# B&R Automation Studio project CNC_Machine_5_18
Automation Studio 4.12.2.93; technology packages: mapp 5.18.0, mappMotion 5.18.1, mappView 5.18.1

## Configuration Config1

CPU X20CP1586, AutomationRuntime C4.73, Build 4.1.2, Vc V4.72.0

### Task classes (Cpu.sw)
```
Cyclic#1:
  Program <- Program.prg
DataObjects: McAcpSys
NcDataObjects: CncProg <- CNCProg.CncProg.dob, McDriveLog
Binaries: McAcpDrv, udbdef, McAcpSim, mvLoader, arflatprv, TCData, OpcUaSrv, McMechSys, FWRules, arcoal, arsvcreg, iomap, asfw, Config_3, Config_4, Role, ashwac, Hierarchy, sysconf, Config_2, arconfig, Config_1, ashwd, Config, User
Libraries: McBase, MpCnc, MpBase, McAxGroup, McPathGen, McAxis, McProgInt, McAcpAx, MpCodeBox, standard, FileIO, AsArLog, AsArProf, AsMem, DataObj, sys_lib, astime, runtime, MpFile, MpServer, MpDatabase, AsHttp, asieccon, asbrstr, asio, asepl, asusb, aruser, arssl, powerlnk, MpData, brsystem, MpAlarmX
```

### Hardware
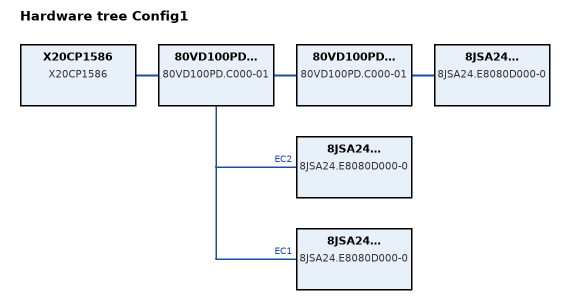
```
80VD100PD.C000-01 : 80VD100PD.C000-01 v2.5.0.0  [PLK1 -> X20CP1586.IF3 [Cable Type=PowerlinkCable, Length=10, Version=1.0.0.3]; PLK2 -> 80VD100PD.C000-01a.PLK2 [Cable Type=PowerlinkCable, Length=10, Version=1.0.0.3]; EC1 -> 8JSA24.E8080D000-0a.EC; EC2 -> 8JSA24.E8080D000-0.EC; MT2 -> 8JSA24.E8080D000-0.MT]
  DriveConfiguration/Module:
    McAcoposTypeID = AcoposMicroDConfig
    ActivateACOPOSSimulationOnPLC = 0
  DriveConfiguration/Channel[1]/RealAxis:
    AxisReference = gAxisQX
    MechanicalElementsIsInvisible = 0
  DriveConfiguration/Channel[1]/RealAxis/MechanicalElements/Gearbox:
    InputIsReadOnly = 0
    Input = 1
    OutputIsReadOnly = 0
    Output = 1
  DriveConfiguration/Channel[1]/RealAxis/MechanicalElements/RotaryToLinearTransformation:
    ReferenceDistanceIsReadOnly = 0
    ReferenceDistance = 1
  DriveConfiguration/Channel[1]/RealAxis/Controller:
    ModeIsReadOnly = 0
    Mode = PositionController
  DriveConfiguration/Channel[1]/RealAxis/Controller/Mode/Position:
    ProportionalGain = 50.0
    IntegrationTime = 0.0
    PredictionTime = 0.0004
    TotalDelayTime = 0.0004
  DriveConfiguration/Channel[1]/RealAxis/Controller/Mode/Speed:
    ProportionalGainIsReadOnly = 0
    ProportionalGain = 2.0
    IntegrationTimeIsReadOnly = 0
    IntegrationTime = 0.0
    FilterTimeIsReadOnly = 0
    FilterTime = 0.0
  DriveConfiguration/Channel[1]/RealAxis/Controller/Mode/LoopFilters:
    LoopFilterXIsReadOnly = 0
    LoopFilter1 = NotUsed
    LoopFilter2 = NotUsed
    LoopFilter3 = NotUsed
  DriveConfiguration/Channel[1]/RealAxis/Homing:
    ModeIsReadOnly = 0
    Mode = Direct
  DriveConfiguration/Channel[1]/RealAxis/Homing/Mode:
    Position = 0.0
    ReferencePulse = NotUsed
  DriveConfiguration/Channel[1]/RealAxis/Homing:
    RestorePositionVariable = 
  DriveConfiguration/Channel[1]/RealAxis/StopReaction:
    QuickstopIsReadOnly = 0
    Quickstop = DecelerationLimit
    DriveErrorIsReadOnly = 0
    DriveError = DecelerationLimit
  DriveConfiguration/Channel[1]/RealAxis/MovementErrorLimits:
    PositionError = 1.0
    VelocityErrorMonitoring = Automatic1
  DriveConfiguration/Channel[1]/RealAxis:
    JerkFilterIsReadOnly = 0
    JerkFilter = NotUsed
  DriveConfiguration/Channel[1]/RealAxis/DigitalInputs/HomingSwitch:
    SourceIsReadOnly = 0
    Source = NotUsed
    Level = High
  DriveConfiguration/Channel[1]/RealAxis/DigitalInputs/PositiveLimitSwitch:
    SourceIsReadOnly = 0
    Source = NotUsed
    Level = High
  DriveConfiguration/Channel[1]/RealAxis/DigitalInputs/NegativeLimitSwitch:
    SourceIsReadOnly = 0
    Source = NotUsed
    Level = High
  DriveConfiguration/Channel[1]/RealAxis/DigitalInputs/Trigger1:
    Source = X2Trigger1
    Level = High
  DriveConfiguration/Channel[1]/RealAxis/DigitalInputs/Trigger2:
    Source = X2Trigger2
    Level = High
  DriveConfiguration/Channel[1]/RealAxis/DigitalInputs/Quickstop:
    Input = Trigger2
  DriveConfiguration/Channel[1]/RealAxis/Simulation:
    SimulationModeOnPLC = SetValueGeneration
    SimulationModeOnACOPOS = NotUsed
  DriveConfiguration/Channel[2]/RealAxis:
    AxisReference = gAxisQY
    MechanicalElementsIsInvisible = 0
  DriveConfiguration/Channel[2]/RealAxis/MechanicalElements/Gearbox:
    InputIsReadOnly = 0
    Input = 1
    OutputIsReadOnly = 0
    Output = 1
  DriveConfiguration/Channel[2]/RealAxis/MechanicalElements/RotaryToLinearTransformation:
    ReferenceDistanceIsReadOnly = 0
    ReferenceDistance = 1
  DriveConfiguration/Channel[2]/RealAxis/Controller:
    ModeIsReadOnly = 0
    Mode = PositionController
  DriveConfiguration/Channel[2]/RealAxis/Controller/Mode/Position:
    ProportionalGain = 50.0
    IntegrationTime = 0.0
    PredictionTime = 0.0004
    TotalDelayTime = 0.0004
  DriveConfiguration/Channel[2]/RealAxis/Controller/Mode/Speed:
    ProportionalGainIsReadOnly = 0
    ProportionalGain = 2.0
    IntegrationTimeIsReadOnly = 0
    IntegrationTime = 0.0
    FilterTimeIsReadOnly = 0
    FilterTime = 0.0
  DriveConfiguration/Channel[2]/RealAxis/Controller/Mode/LoopFilters:
    LoopFilterXIsReadOnly = 0
    LoopFilter1 = NotUsed
    LoopFilter2 = NotUsed
    LoopFilter3 = NotUsed
  DriveConfiguration/Channel[2]/RealAxis/Homing:
    ModeIsReadOnly = 0
    Mode = Direct
  DriveConfiguration/Channel[2]/RealAxis/Homing/Mode:
    Position = 0.0
    ReferencePulse = NotUsed
  DriveConfiguration/Channel[2]/RealAxis/Homing:
    RestorePositionVariable = 
  DriveConfiguration/Channel[2]/RealAxis/StopReaction:
    QuickstopIsReadOnly = 0
    Quickstop = DecelerationLimit
    DriveErrorIsReadOnly = 0
    DriveError = DecelerationLimit
  DriveConfiguration/Channel[2]/RealAxis/MovementErrorLimits:
    PositionError = 1.0
    VelocityErrorMonitoring = Automatic1
  DriveConfiguration/Channel[2]/RealAxis:
    JerkFilterIsReadOnly = 0
    JerkFilter = NotUsed
  DriveConfiguration/Channel[2]/RealAxis/DigitalInputs/HomingSwitch:
    SourceIsReadOnly = 0
    Source = NotUsed
    Level = High
  DriveConfiguration/Channel[2]/RealAxis/DigitalInputs/PositiveLimitSwitch:
    SourceIsReadOnly = 0
    Source = NotUsed
    Level = High
  DriveConfiguration/Channel[2]/RealAxis/DigitalInputs/NegativeLimitSwitch:
    SourceIsReadOnly = 0
    Source = NotUsed
    Level = High
  DriveConfiguration/Channel[2]/RealAxis/DigitalInputs/Trigger1:
    Source = X2Trigger1
    Level = High
  DriveConfiguration/Channel[2]/RealAxis/DigitalInputs/Trigger2:
    Source = X2Trigger2
    Level = High
  DriveConfiguration/Channel[2]/RealAxis/DigitalInputs/Quickstop:
    Input = Trigger2
  DriveConfiguration/Channel[2]/RealAxis/Simulation:
    SimulationModeOnPLC = SetValueGeneration
    SimulationModeOnACOPOS = NotUsed
80VD100PD.C000-01a : 80VD100PD.C000-01 v2.5.0.0  [PLK2 -> 80VD100PD.C000-01.PLK2 [Cable Type=PowerlinkCable, Length=10, Version=1.0.0.3]; EC1 -> 8JSA24.E8080D000-0b.EC]
  DriveConfiguration/Module:
    McAcoposTypeID = AcoposMicroDConfig
    ActivateACOPOSSimulationOnPLC = 0
  DriveConfiguration/Channel[1]/RealAxis:
    AxisReference = gAxisQZ
    MechanicalElementsIsInvisible = 0
  DriveConfiguration/Channel[1]/RealAxis/MechanicalElements/Gearbox:
    InputIsReadOnly = 0
    Input = 1
    OutputIsReadOnly = 0
    Output = 1
  DriveConfiguration/Channel[1]/RealAxis/MechanicalElements/RotaryToLinearTransformation:
    ReferenceDistanceIsReadOnly = 0
    ReferenceDistance = 1
  DriveConfiguration/Channel[1]/RealAxis/Controller:
    ModeIsReadOnly = 0
    Mode = PositionController
  DriveConfiguration/Channel[1]/RealAxis/Controller/Mode/Position:
    ProportionalGain = 50.0
    IntegrationTime = 0.0
    PredictionTime = 0.0004
    TotalDelayTime = 0.0004
  DriveConfiguration/Channel[1]/RealAxis/Controller/Mode/Speed:
    ProportionalGainIsReadOnly = 0
    ProportionalGain = 2.0
    IntegrationTimeIsReadOnly = 0
    IntegrationTime = 0.0
    FilterTimeIsReadOnly = 0
    FilterTime = 0.0
  DriveConfiguration/Channel[1]/RealAxis/Controller/Mode/LoopFilters:
    LoopFilterXIsReadOnly = 0
    LoopFilter1 = NotUsed
    LoopFilter2 = NotUsed
    LoopFilter3 = NotUsed
  DriveConfiguration/Channel[1]/RealAxis/Homing:
    ModeIsReadOnly = 0
    Mode = Direct
  DriveConfiguration/Channel[1]/RealAxis/Homing/Mode:
    Position = 0.0
    ReferencePulse = NotUsed
  DriveConfiguration/Channel[1]/RealAxis/Homing:
    RestorePositionVariable = 
  DriveConfiguration/Channel[1]/RealAxis/StopReaction:
    QuickstopIsReadOnly = 0
    Quickstop = DecelerationLimit
    DriveErrorIsReadOnly = 0
    DriveError = DecelerationLimit
  DriveConfiguration/Channel[1]/RealAxis/MovementErrorLimits:
    PositionError = 1.0
    VelocityErrorMonitoring = Automatic1
  DriveConfiguration/Channel[1]/RealAxis:
    JerkFilterIsReadOnly = 0
    JerkFilter = NotUsed
  DriveConfiguration/Channel[1]/RealAxis/DigitalInputs/HomingSwitch:
    SourceIsReadOnly = 0
    Source = NotUsed
    Level = High
  DriveConfiguration/Channel[1]/RealAxis/DigitalInputs/PositiveLimitSwitch:
    SourceIsReadOnly = 0
    Source = NotUsed
    Level = High
  DriveConfiguration/Channel[1]/RealAxis/DigitalInputs/NegativeLimitSwitch:
    SourceIsReadOnly = 0
    Source = NotUsed
    Level = High
  DriveConfiguration/Channel[1]/RealAxis/DigitalInputs/Trigger1:
    Source = X2Trigger1
    Level = High
  DriveConfiguration/Channel[1]/RealAxis/DigitalInputs/Trigger2:
    Source = X2Trigger2
    Level = High
  DriveConfiguration/Channel[1]/RealAxis/DigitalInputs/Quickstop:
    Input = Trigger2
  DriveConfiguration/Channel[1]/RealAxis/Simulation:
    SimulationModeOnPLC = SetValueGeneration
    SimulationModeOnACOPOS = NotUsed
  DriveConfiguration/Channel[2]/RealAxis:
    AxisReference = 
    MechanicalElementsIsInvisible = 0
  DriveConfiguration/Channel[2]/RealAxis/MechanicalElements/Gearbox:
    InputIsReadOnly = 0
    Input = 1
    OutputIsReadOnly = 0
    Output = 1
  DriveConfiguration/Channel[2]/RealAxis/MechanicalElements/RotaryToLinearTransformation:
    ReferenceDistanceIsReadOnly = 0
    ReferenceDistance = 1
  DriveConfiguration/Channel[2]/RealAxis/Controller:
    ModeIsReadOnly = 0
    Mode = PositionController
  DriveConfiguration/Channel[2]/RealAxis/Controller/Mode/Position:
    ProportionalGain = 50.0
    IntegrationTime = 0.0
    PredictionTime = 0.0004
    TotalDelayTime = 0.0004
  DriveConfiguration/Channel[2]/RealAxis/Controller/Mode/Speed:
    ProportionalGainIsReadOnly = 0
    ProportionalGain = 2.0
    IntegrationTimeIsReadOnly = 0
    IntegrationTime = 0.0
    FilterTimeIsReadOnly = 0
    FilterTime = 0.0
  DriveConfiguration/Channel[2]/RealAxis/Controller/Mode/LoopFilters:
    LoopFilterXIsReadOnly = 0
    LoopFilter1 = NotUsed
    LoopFilter2 = NotUsed
    LoopFilter3 = NotUsed
  DriveConfiguration/Channel[2]/RealAxis/Homing:
    ModeIsReadOnly = 0
    Mode = Direct
  DriveConfiguration/Channel[2]/RealAxis/Homing/Mode:
    Position = 0.0
    ReferencePulse = NotUsed
  DriveConfiguration/Channel[2]/RealAxis/Homing:
    RestorePositionVariable = 
  DriveConfiguration/Channel[2]/RealAxis/StopReaction:
    QuickstopIsReadOnly = 0
    Quickstop = DecelerationLimit
    DriveErrorIsReadOnly = 0
    DriveError = DecelerationLimit
  DriveConfiguration/Channel[2]/RealAxis/MovementErrorLimits:
    PositionError = 1.0
    VelocityErrorMonitoring = Automatic1
  DriveConfiguration/Channel[2]/RealAxis:
    JerkFilterIsReadOnly = 0
    JerkFilter = NotUsed
  DriveConfiguration/Channel[2]/RealAxis/DigitalInputs/HomingSwitch:
    SourceIsReadOnly = 0
    Source = NotUsed
    Level = High
  DriveConfiguration/Channel[2]/RealAxis/DigitalInputs/PositiveLimitSwitch:
    SourceIsReadOnly = 0
    Source = NotUsed
    Level = High
  DriveConfiguration/Channel[2]/RealAxis/DigitalInputs/NegativeLimitSwitch:
    SourceIsReadOnly = 0
    Source = NotUsed
    Level = High
  DriveConfiguration/Channel[2]/RealAxis/DigitalInputs/Trigger1:
    Source = X2Trigger1
    Level = High
  DriveConfiguration/Channel[2]/RealAxis/DigitalInputs/Trigger2:
    Source = X2Trigger2
    Level = High
  DriveConfiguration/Channel[2]/RealAxis/DigitalInputs/Quickstop:
    Input = Trigger2
  DriveConfiguration/Channel[2]/RealAxis/Simulation:
    SimulationModeOnPLC = SetValueGeneration
    SimulationModeOnACOPOS = NotUsed
8JSA24.E8080D000-0 : 8JSA24.E8080D000-0 v1.0.6.30  [EC -> 80VD100PD.C000-01.EC2; MT -> 80VD100PD.C000-01.MT2]
8JSA24.E8080D000-0a : 8JSA24.E8080D000-0 v1.0.6.30  [EC -> 80VD100PD.C000-01.EC1; MT -> 80VD100PD.C000-01.MT1]
8JSA24.E8080D000-0b : 8JSA24.E8080D000-0 v1.0.6.30  [EC -> 80VD100PD.C000-01a.EC1; MT -> 80VD100PD.C000-01a.MT1]
X20CP1586 : X20CP1586 v1.10.0.0
  Connector IF1:
    ActivateIna = 0
  Connector IF2:
    ActivateDevice = 1
    InaPort = 11160
  Connector IF3:
    DNAConfiguration = manual
  ConfigurationID = CNC_Machine_5_18_Config1
  Simulation = 1
  TimerDeviceType = EPLX2X
  TimerDevice = X20CP1586.IF3
  TaskClassIdleTime = 2000
  Cyclic1Tolerance = 0
  FileDevice1
  FileDeviceName1 = HD
  FileDevicePath1 = C:\CNC\
  ActivateOpcUa = 1
  OpcUaInformationModels_PV_Version = 1
```

### Config_1.axesgroup - X20CP1586/mappMotion/3AxesCNCXYZ/Config_1.axesgroup
```
Element gCncXYZ (Type=axesgroup)
  Type = PathGenAxesGroup
    ProcessingTaskClass = 255
    License = 1
    PhysicalAxes:
      JointAxes:
        JointAxisAxisRefIsReadOnly = 0
        JointAxis[1]:
          Name = QX
          AxisRef = gAxisQX
        JointAxis[2]:
          Name = QY
          AxisRef = gAxisQY
        JointAxis[3]:
          Name = QZ
          AxisRef = gAxisQZ
    MechanicalSystem:
      MechSysRefIsReadOnly = 0
      MechSysRef = MechSys_3AxCNCXYZ
    BasicSettings:
      ModalDataBehaviour = ResetToDefault
      GeometryPlanning:
        TCPResolutionIsReadOnly = 0
        TCPResolution:
          LengthResolution = 0.001
          AngleResolution = 0.001
        RoundingMode = Standard
        MaxCornerDeviation = 0.0
        MaxTangentialTransitionDeviation = 0.0
        MaxRadiusDeviation = 0.001
        WorkingPlane = XY
      TrajectoryPlanningIsReadOnly = 0
      TrajectoryPlanning = Basic
        LimitCheckResolutionIsReadOnly = 0
        LimitCheckResolution = UserDefinedTime
          TimeIsReadOnly = 0
          Time = 0.01
        BufferTime = UserDefinedTime
          Time = 0.1
      Miscellaneous:
        NonMovementsLimit = NotUsed
    AxesGroupFeatures:
      FeatureRef[1] = Feature_Programs
      FeatureRef[2] = Feature_Jogging
  Alarms = MpAlarmX
```

### Config_2.axis - X20CP1586/mappMotion/3AxesCNCXYZ/Config_2.axis
```
Element gAxisQX (Type=axis)
  BaseTypeIsReadOnly = 0
  BaseType = LinearBounded
    MeasurementUnit = 5066068
    MeasurementResolutionIsReadOnly = 0
    MeasurementResolution = 0.01
    CountDirectionIsReadOnly = 0
    CountDirection = Standard
  MovementLimitsIsReadOnly = 0
  MovementLimits = Internal
    Position:
      LowerLimitMin = -1.79769313486231E308
      UpperLimitMax = 1.79769313486231E308
      LowerLimit = -1000.0
      UpperLimit = 1000.0
    VelocityIsReadOnly = 0
    Velocity:
      VelocityMax = 3.4E38
      Velocity = 10.0
    AccelerationIsReadOnly = 0
    Acceleration:
      AccelerationMax = 3.4E38
      Acceleration = 50.0
    DecelerationIsReadOnly = 0
    Deceleration:
      DecelerationMax = 3.4E38
      Deceleration = 50.0
  Alarms = None
Element gAxisQY (Type=axis)
  BaseTypeIsReadOnly = 0
  BaseType = LinearBounded
    MeasurementUnit = 5066068
    MeasurementResolutionIsReadOnly = 0
    MeasurementResolution = 0.01
    CountDirectionIsReadOnly = 0
    CountDirection = Standard
  MovementLimitsIsReadOnly = 0
  MovementLimits = Internal
    Position:
      LowerLimitMin = -1.79769313486231E308
      UpperLimitMax = 1.79769313486231E308
      LowerLimit = -1000.0
      UpperLimit = 1000.0
    VelocityIsReadOnly = 0
    Velocity:
      VelocityMax = 3.4E38
      Velocity = 10.0
    AccelerationIsReadOnly = 0
    Acceleration:
      AccelerationMax = 3.4E38
      Acceleration = 50.0
    DecelerationIsReadOnly = 0
    Deceleration:
      DecelerationMax = 3.4E38
      Deceleration = 50.0
  Alarms = None
Element gAxisQZ (Type=axis)
  BaseTypeIsReadOnly = 0
  BaseType = LinearBounded
    MeasurementUnit = 5066068
    MeasurementResolutionIsReadOnly = 0
    MeasurementResolution = 0.01
    CountDirectionIsReadOnly = 0
    CountDirection = Standard
  MovementLimitsIsReadOnly = 0
  MovementLimits = Internal
    Position:
      LowerLimitMin = -1.79769313486231E308
      UpperLimitMax = 1.79769313486231E308
      LowerLimit = -1000.0
      UpperLimit = 1000.0
    VelocityIsReadOnly = 0
    Velocity:
      VelocityMax = 3.4E38
      Velocity = 10.0
    AccelerationIsReadOnly = 0
    Acceleration:
      AccelerationMax = 3.4E38
      Acceleration = 50.0
    DecelerationIsReadOnly = 0
    Deceleration:
      DecelerationMax = 3.4E38
      Deceleration = 50.0
  Alarms = None
```

### Config_3.mechanicalsystem - X20CP1586/mappMotion/3AxesCNCXYZ/Config_3.mechanicalsystem
```
Element MechSys_3AxCNCXYZ (Type=mechanicalsystem)
  TypeIsReadOnly = 0
  Type = 3AxesCNC
    Subtype = 3AxesCNCXYZ
      CoordinatesNames = Default
        XCoordinateName = X
        YCoordinateName = Y
        ZCoordinateName = Z
      WireFrameModel = Standard
        FlangeToTcp = ConnectionLine
          DistanceMin = -1.79769313486231E308
          DistanceMax = 1.79769313486231E308
          Distance = 0.0
      JointAxesPositionLimits:
        JointAxisIsReadOnly = 0
        JointAxis[1] = UseAxisLimits
        JointAxis[2] = UseAxisLimits
        JointAxis[3] = UseAxisLimits
```

### Config_4.axesgroupfeature - X20CP1586/mappMotion/3AxesCNCXYZ/Config_4.axesgroupfeature
```
Element Feature_Programs (Type=axesgroupfeature)
  Type = Program
    ModalDataBehaviour = UseAxesGroupSettings
    InitialSettings:
      InterpolationTypes = LinearRapid
      PositionCoordinates = Absolute
      CircleCoordinates = Relative
      JACS_ACSProgramming = JACS
      ContourConnection = Inactive
      ProgrammingUnits = UseAxesGroupSettings
      Feedrates:
        FeedPath = Standard
        FeedCharacteristic = StandardCharacteristic
        FeedType = Feedrate
        FeedReduction = Inactive
        FeedrateValue = 0.0
        InverseFeedrateValue = 0.0
        FeedratePerRevValue = 0.0
    DefaultLanguage = BRGCode
    Location = Default
      FileDevice = CNC_PrgDir
Element Feature_Jogging (Type=axesgroupfeature)
  Type = Jogging
```

### Config_5.mpfilemanager - X20CP1586/mappServices/Config_5.mpfilemanager
```
Element FileManagement (Type=mpfilemanager)
  FileManager:
    Devices:
      0:
        DeviceName = HD
        Text = Festplatte
      1:
        DeviceName = 
        Text = 
    Access:
      0:
        Folder = *
        Roles:
          0:
            Role = Everyone
            Rights:
              Visible = TRUE
              FolderRead = TRUE
              FileRead = TRUE
              FileEdit = TRUE
              FolderEdit = TRUE
          1:
            Role = Administrators
            Rights:
              Visible = TRUE
              FolderRead = TRUE
              FileRead = TRUE
              FileEdit = TRUE
              FolderEdit = TRUE
```

### Config_6.mpalarmxcore - X20CP1586/mappServices/Config_6.mpalarmxcore
```
Element gAlarmXCore (Type=mpalarmxcore)
  mapp.AlarmX.Core.Configuration:
    [0]:
      Name = limitX
      Message = {$IAT/AlarmList/limitX}: {&actPosX}
      Code = 1234
      Severity = 10
    [1]:
      Name = limitY
      Message = {$IAT/AlarmList/limitY}: {&actPosY}
      Code = 1235
      Severity = 10
    [2]:
      Name = limitZ
      Message = {$IAT/AlarmList/limitZ}: {&actPosZ}
      Code = 1236
      Severity = 10
  mapp.AlarmX.Core.Snippets:
    [0]:
      Key = actPosX
      Value:
        PV = ::Program:CncMachine.X
    [1]:
      Key = actPosY
      Value:
        PV = ::Program:CncMachine.Y
    [2]:
      Key = actPosZ
      Value:
        PV = ::Program:CncMachine.Z
```

## Logical view

Binary libraries used (declarations not repeated): operator, runtime, astime, AsIecCon, McBase 5.18.1, MpCnc 5.18.1, MpBase 5.18.0, McAxGroup 5.18.1, McPathGen 5.18.1, McAxis 5.18.1, McProgInt 5.18.1, McAcpAx 5.18.1, MpCodeBox 5.18.0, standard, FileIO, AsArLog, AsArProf, AsMem, DataObj, sys_lib, MpFile, MpServer, MpDatabase 5.18.0, AsHttp, MpData, brsystem, MpAlarmX


### Program Logical/Program (IEC)

#### Variables.var
```iecst
VAR
	CncMachineParam : MpCnc3AxisParType;
	CncMachine : MpCnc3Axis;
	fileManagerSetup : MpFileManagerUISetupType;
	fileManagerConnect : MpFileManagerUIConnectType;
	fileManagerConfig : MpFileManagerConfig;
	fileManager : MpFileManagerUI;
	mpDataRegZ : MpDataRegPar;
	mpDataRegY : MpDataRegPar;
	mpDataRegX : MpDataRegPar;
	mpDataRecorderFB : MpDataRecorder;
	enableControl : BOOL;
	btnIsOnOff : STRING[20];
	ledPowerOn : STRING[20];
	ledIsHome : STRING[20];
	ledIsError : STRING[20];
	speedFactor : UINT;
	mpAlarm : MpAlarmXCore;
	acknowledge : BOOL;
	reset : BOOL;
	endStopReachedX : BOOL;
	endStopReachedY : BOOL;
	endStopReachedZ : BOOL;
	XMinLimit : REAL;
	XMaxLimit : REAL;
	YMinLimit : REAL;
	YMaxLimit : REAL;
	ZMinLimit : REAL;
	ZMaxLimit : REAL;
	xLimitAlarmActive : BOOL;
	zLimitAlarmActive : BOOL;
	yLimitAlarmActive : BOOL;
END_VAR
```

#### Main.st
```iecst
PROGRAM _INIT
	enableControl := TRUE;
	speedFactor := 1;

	CncMachine.Enable := TRUE;

	CncMachine.Override := 100;
	CncMachineParam.ProgramName := 'CncProg';

	mpDataRecorderFB.Enable := TRUE;
	mpDataRecorderFB.DeviceName := ADR('HD');
	mpDataRecorderFB.MpLink := ADR(gDataRecorder);
	mpDataRecorderFB.RecordMode := mpDATA_RECORD_MODE_VALUE;

	mpDataRegX.Enable := TRUE;
	mpDataRegX.MpLink := ADR(gDataRecorder);
	mpDataRegX.PVName := ADR('::Program:CncMachine.X');

	mpDataRegY.Enable := TRUE;
	mpDataRegY.MpLink := ADR(gDataRecorder);
	mpDataRegY.PVName := ADR('::Program:CncMachine.Y');

	mpDataRegZ.Enable := TRUE;
	mpDataRegZ.MpLink := ADR(gDataRecorder);
	mpDataRegZ.PVName := ADR('::Program:CncMachine.Z');

	mpAlarm.Enable := TRUE;
	mpAlarm.MpLink := ADR(gAlarmXCore);

	XMinLimit := -50;
	XMaxLimit := 50;
	YMinLimit := -50;
	YMaxLimit := 50;
	ZMinLimit := -50;
	ZMaxLimit := 50;

END_PROGRAM

PROGRAM _CYCLIC
	CncMachine.MpLink := ADR(gCncXYZ);
	CncMachine.Parameters := ADR(CncMachineParam);
	CncMachine();

	mpAlarm();

	mpDataRecorderFB();
	mpDataRegX();
	mpDataRegY();
	mpDataRegZ();

	IF CncMachine.PowerOn THEN
		ledPowerOn := 'Solid_Gray_Green';
		btnIsOnOff := 'Off';
	ELSE
		ledPowerOn := 'Solid_Gray_Gray';
		btnIsOnOff := 'On';
	END_IF

	IF CncMachine.IsHomed THEN
		ledIsHome := 'Solid_Gray_Green';
	ELSE
		ledIsHome := 'Solid_Gray_Gray';
	END_IF

	IF CncMachine.Error THEN
		ledIsError := 'Solid_Gray_Red';
	ELSE
		ledIsError := 'Solid_Gray_Green';
	END_IF

	IF CncMachine.X < XMinLimit OR CncMachine.X > XMaxLimit THEN
		IF xLimitAlarmActive = FALSE THEN
			MpAlarmXSet(gAlarmXCore,'limitX');
			xLimitAlarmActive := TRUE;
		END_IF
		IF (CncMachine.X < XMinLimit AND CncMachineParam.Jog.Velocity[0] <= 0)
			OR (CncMachine.X > XMaxLimit AND CncMachineParam.Jog.Velocity[0] >= 0) THEN
			CncMachineParam.Jog.Velocity[0] := 0;
			endStopReachedX := TRUE;
		END_IF
	ELSE
		endStopReachedX := FALSE;
		xLimitAlarmActive := FALSE;
	END_IF

	IF acknowledge THEN
		MpAlarmXAcknowledge(gAlarmXCore,'limitX');
	END_IF

	IF reset THEN
		MpAlarmXReset(gAlarmXCore,'limitX');
	END_IF

	IF CncMachine.Y < YMinLimit OR CncMachine.Y > YMaxLimit THEN
		IF yLimitAlarmActive = FALSE THEN
			MpAlarmXSet(gAlarmXCore,'limitY');
			yLimitAlarmActive := TRUE;
		END_IF
		IF (CncMachine.Y < YMinLimit AND CncMachineParam.Jog.Velocity[1] <= 0)
			OR (CncMachine.Y > YMaxLimit AND CncMachineParam.Jog.Velocity[1] >= 0) THEN
			CncMachineParam.Jog.Velocity[1] := 0;
			endStopReachedY := TRUE;
		END_IF
	ELSE
		endStopReachedY := FALSE;
		yLimitAlarmActive := FALSE;
	END_IF

	IF acknowledge THEN
		MpAlarmXAcknowledge(gAlarmXCore,'limitY');
	END_IF

	IF reset THEN
		MpAlarmXReset(gAlarmXCore,'limitY');
	END_IF

	IF CncMachine.Z < ZMinLimit OR CncMachine.Z > ZMaxLimit THEN
		IF zLimitAlarmActive = FALSE THEN
			MpAlarmXSet(gAlarmXCore,'limitZ');
			zLimitAlarmActive := TRUE;
		END_IF
		IF (CncMachine.Z < ZMinLimit AND CncMachineParam.Jog.Velocity[2] <= 0)
				OR (CncMachine.Z > ZMaxLimit AND CncMachineParam.Jog.Velocity[2] >= 0) THEN
			CncMachineParam.Jog.Velocity[2] := 0;
			endStopReachedZ := TRUE;
		END_IF
	ELSE
		endStopReachedZ := FALSE;
		zLimitAlarmActive := FALSE;
	END_IF

	IF acknowledge THEN
		MpAlarmXAcknowledge(gAlarmXCore,'limitZ');
	END_IF

	IF reset THEN
		MpAlarmXReset(gAlarmXCore,'limitZ');
	END_IF

END_PROGRAM

PROGRAM _EXIT

END_PROGRAM
```

### Data object Logical/CNCProg/CncProg (Cnc)

#### CncProg.cnc
```
%001 (CncProgram)

N10 G90     (absolute coordinates)
N20 F300    (Feed rate in measurements units/min)

N30 G04 2   (dwell time 2s)

N50 G01 X80 Y100  (linear move)

N60 G04 2         (dwell time 2s)

N100 G00 X0 Y0    (rapid move to zero)
N999 M30
```

- Visualisation Logical/mappView (not shown)

Listed in the project but not available here: Logical/Global.typ, Logical/Global.var
